(* PLC project Unnamed, Unknown Unnamed 1 *)
(* stored: creationDateTime 2021-03-11T20:50:13, modificationDateTime 2023-08-05T13:26:45 *)

PROGRAM Main
  VAR
    I_PbFill AT %IX100.0 : BOOL;  (* Pushbutton Fill button (Normal Open NO) *)
    I_PbDischarge AT %IX100.1 : BOOL := True;  (* Pushbutton Discharge button (Normal Clossed NC) *)
    Q_FillValve AT %QX100.0 : BOOL;
    Q_FillLight AT %QX100.1 : BOOL;
    Q_DischargeValve AT %QX100.2 : BOOL;
    Q_LightDischarge AT %QX100.3 : BOOL;
    Q_Display AT %QW100 : INT;
  END_VAR
  VAR
    Filling : BOOL;
    Discharging : BOOL;
    TimeFilling : TIME;
    TimeFillingInt : INT;
    TimeDischarging : TIME;
    TimeDischargingInt : INT;
    TON0 : TON;
    RS0 : RS;
    R_TRIG0 : R_TRIG;
    TON1 : TON;
    RS1 : RS;
    F_TRIG0 : F_TRIG;
    Placeholder : INT;
  END_VAR
  VAR
    Simulation AT %QW101 : INT;
  END_VAR

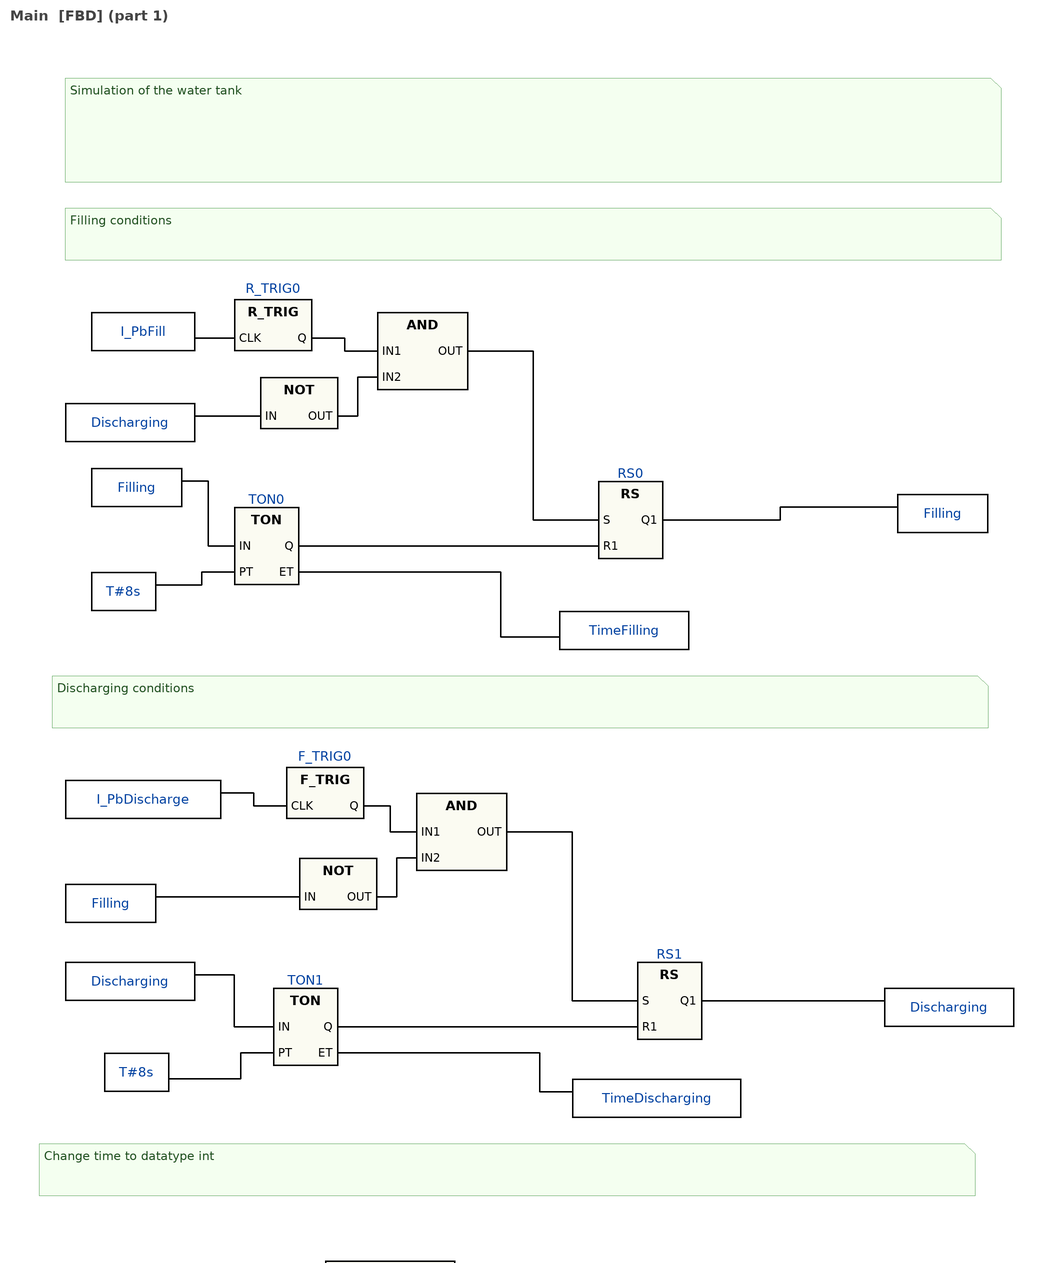
(* FBD diagram, written out as Structured Text *)
(* Simulation of the water tank *)
(* Filling conditions *)
R_TRIG0(CLK := I_PbFill);
TON0(IN := Filling, PT := T#8s);
RS0(S := R_TRIG0.Q AND NOT Discharging, R1 := TON0.Q);
Filling := RS0.Q1;
TimeFilling := TON0.ET;
(* Discharging conditions *)
F_TRIG0(CLK := I_PbDischarge);
TON1(IN := Discharging, PT := T#8s);
RS1(S := F_TRIG0.Q AND NOT Filling, R1 := TON1.Q);
Discharging := RS1.Q1;
TimeDischarging := TON1.ET;
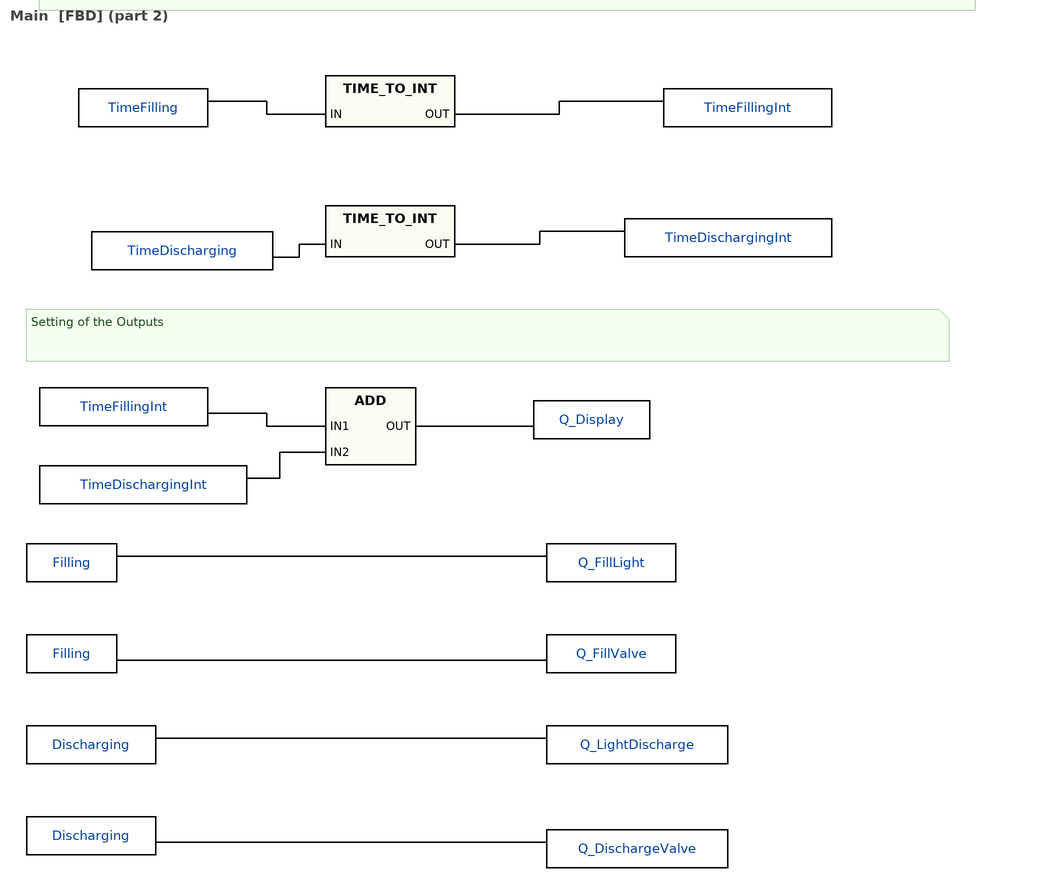
(* Change time to datatype int *)
TimeFillingInt := TIME_TO_INT(TimeFilling);
TimeDischargingInt := TIME_TO_INT(TimeDischarging);
(* Setting of the Outputs *)
Q_Display := TimeFillingInt + TimeDischargingInt;
Q_FillLight := Filling;
Q_FillValve := Filling;
Q_LightDischarge := Discharging;
Q_DischargeValve := Discharging;
END_PROGRAM

CONFIGURATION Config0
  RESOURCE Res0 ON PLC
    TASK task0(INTERVAL := T#20ms, PRIORITY := 0);
    PROGRAM instance0 WITH task0 : Main;
  END_RESOURCE
END_CONFIGURATION
